# EPICS substitutions: iocBoot/iocScanLib/scanLib.substitutions
file "$(TOP)/db/scanLib.template"
{
pattern
{  P,        R,      TOMOSCAN_PREFIX,  INSITU_PV, SAMPLE_X, SAMPLE_Y}
{2bmb:, ScanLib:,     2bmb:TomoScan:     2bm:m1,  2bmb:m63, 2bmb:m25}
}
